// TIA Portal project "SCL" (V19)

(* hardware
DEVICE "S7-1500/ET200MP station_1"  S7-1500 station
   slot 0: "Rail_0"  Rack  6ES7 590-1***0-0AA0
   slot 1: "PLC_1"  CPU 1513-1 PN  6ES7 513-1AL02-0AB0  V2.9
      slot 3: "CPU display_1"  6ES7591-1AA00-0AA0
      slot 32768: "PROFINET interface_1"  X1
         slot 32769: "Port_1"  X1 P1
         slot 32770: "Port_2"  X1 P2
      slot 34817: "Virtual CP interface port_1"  Virtual CP interface port  Virtual CP interface port
   slot 2: "DI 16x24VDC BA_1"  DI 16x24VDC BA  6ES7 521-1BH10-0AA0  V1.1
   slot 3: "DQ 16x24VDC/0.5A BA_1"  DQ 16x24VDC/0.5A BA  6ES7 522-1BH10-0AA0  V1.1
*)

// ===== PLC "PLC_1"  CPU 1513-1 PN =====

VAR_GLOBAL   // PLC tag table "Default tag table"
   "At Entry" AT %I0.0 : Bool;
   "At Load" AT %I0.1 : Bool;
   "At left" AT %I0.2 : Bool;
   "At Middle" AT %I0.3 : Bool;
   "At Right" AT %I0.4 : Bool;
   "At Unload" AT %I0.5 : Bool;
   "At Exit" AT %I0.6 : Bool;
   "Moving X" AT %I0.7 : Bool;
   "Moving Z" AT %I1.0 : Bool;
   "Start" AT %I1.1 : Bool;
   "Reset" AT %I1.2 : Bool;
   "Stop" AT %I1.3 : Bool;
   "Emergency stop" AT %I1.4 : Bool;
   "Auto" AT %I1.5 : Bool;
   "FACTORY I/O (Runing)" AT %I1.6 : Bool;
   "Entry Conveyor" AT %Q0.0 : Bool;
   "Load Conveyor" AT %Q0.1 : Bool;
   "Forks Left" AT %Q0.2 : Bool;
   "Forks Right" AT %Q0.3 : Bool;
   "Lift" AT %Q0.4 : Bool;
   "Unload Conveyor" AT %Q0.5 : Bool;
   "Exit Conveyor" AT %Q0.6 : Bool;
   "Start light" AT %Q0.7 : Bool;
   "Reset light" AT %Q1.0 : Bool;
   "Stop light" AT %Q1.1 : Bool;
   "Target position" AT %QW30 : Int;
   "State0" AT %M0.0 : Bool;
   "State1" AT %M0.1 : Bool;
   "State2" AT %M0.2 : Bool;
   "State3" AT %M0.3 : Bool;
   "State4" AT %M0.4 : Bool;
   "State5" AT %M0.5 : Bool;
   "State6" AT %M0.6 : Bool;
   "State7" AT %M0.7 : Bool;
   "State8" AT %M1.0 : Bool;
   "State9" AT %M1.1 : Bool;
   "Tag_1" AT %M1.3 : Bool;
   "Tag_2" AT %M1.4 : Bool;
   "Tag_3" AT %M1.5 : Bool;
   "Tag_4" AT %M1.6 : Bool;
   "Tag_5" AT %M1.2 : Bool;
   "t" AT %MW30 : Int;
   "Tag_6" AT %M1.7 : Bool;
   "case" AT %MW2 : Int;
END_VAR

FUNCTION "Block_1" : Void   // FC1, SCL
{ S7_Optimized_Access := 'TRUE' }
VERSION : 0.1
BEGIN
   IF "Start light" THEN

       // Statement section IF
       CASE "case" OF
           0:  // Statement section case 1
               "Entry Conveyor" := FALSE;
               "Load Conveyor" := FALSE;
               "Forks Left" := FALSE;
               "Forks Right" := FALSE;
               "Lift" := FALSE;
               "Unload Conveyor" := FALSE;
               "Exit Conveyor" := FALSE;
               "case" := 1;

           1:  // Statement section case 2 to 4
               "Entry Conveyor" := TRUE;
               "Load Conveyor" := TRUE;
               IF NOT "At Load" THEN
                   // Statement section IF
                   "case" := 2;
               END_IF;
           2:
               "Forks Left" := 1;
               "Entry Conveyor" := 0;
               "Load Conveyor" := 0;
               IF "At left" THEN
                   // Statement section IF
                   "case" := 3;
               END_IF;
           3:
               "Lift" := 1;
               "R_TRIG_DB"(CLK:="Moving Z",
                           Q=>"Tag_1");

               IF "Tag_1" THEN
                   // Statement section IF
                   "case" := 4;
               END_IF;

           4:
               "Forks Left" := 0;
               IF "At Middle" THEN
                   // Statement section IF
                   "case" := 5;
               END_IF;
               "Tag_5" := 1;
           5:


               //"R_TRIG_DB_1"(CLK:="Tag_5",
                             //Q=>"Tag_6");
               //IF "Tag_5" THEN
                   // Statement section IF
                  // "Tag_5" := FALSE;
                  // "Target position" := "t";
                  // "t" := "t" + 1;


              // END_IF;
               WHILE "Tag_5" DO
                   // Statement section WHILE
                   "Tag_5" := FALSE;
                   "Target position" := "t";
                   "t" := "t" + 1;;
               END_WHILE;



               "F_TRIG_DB"(CLK:="Moving Z",
                           Q=>"Tag_2");

               "F_TRIG_DB_1"(CLK:="Moving X",
                             Q=>"Tag_3");

               IF ("Tag_2" AND NOT "Moving X") OR ("Tag_3" AND NOT "Moving Z") THEN
                   // Statement section IF

                   "case":=6;
               END_IF;

           6:

               "Forks Right" := 1;
               IF "At Right" THEN
                   // Statement section IF
                   "case" := 7;
               END_IF;
           7:
               "Lift" := 0
               ;
               "F_TRIG_DB_2"(CLK:="Moving Z",
                             Q=>"Tag_4");
               IF "Tag_4" THEN
                   // Statement section IF
                   "case" := 8;
               END_IF;
           8:
               "Forks Right" := 0;
               IF "At Middle" THEN
                   // Statement section IF
                   "case":=9;
               END_IF;
           9:
               "Target position" := 55;
               "case" := 0;


       END_CASE;

       ;
   END_IF;
END_FUNCTION

FUNCTION "Block_2" : Void   // FC2, LAD
{ S7_Optimized_Access := 'TRUE' }
VERSION : 0.1
BEGIN

REGION Network 1
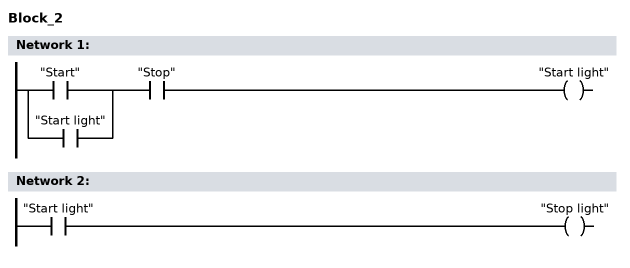
   RUNG wire#powerrail
      Contact( "Start" )
      wire#w1
      Contact( "Stop" )
      Coil( "Start light" )
   END_RUNG
   RUNG wire#powerrail
      Contact( "Start light" )
   END_RUNG wire#w1
   // the same network as SCL:
   "Start light" := ("Start" OR "Start light") AND "Stop";
END_REGION

REGION Network 2
   RUNG wire#powerrail
      Contact( "Start light" )
      Coil( "Stop light" )
   END_RUNG
   // the same network as SCL:
   "Stop light" := "Start light";
END_REGION
END_FUNCTION

ORGANIZATION_BLOCK "Main"   // OB1, LAD, ProgramCycle
TITLE = "Main Program Sweep (Cycle)"
{ S7_Optimized_Access := 'TRUE' }
VERSION : 0.1
   VAR_INPUT
      Initial_Call : Bool;   // Initial call of this OB
      Remanence : Bool;   // =True, if remanent data are available
   END_VAR
BEGIN

REGION Network 1
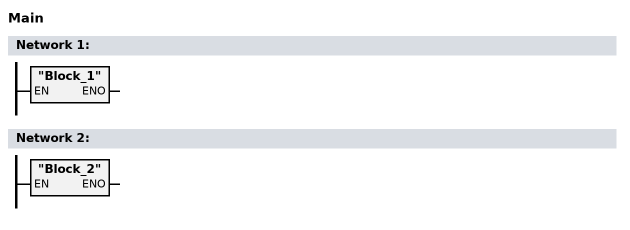
   RUNG wire#powerrail
      "Block_1"()
   END_RUNG
   // the same network as SCL:
   "Block_1"();
END_REGION

REGION Network 2
   RUNG wire#powerrail
      "Block_2"()
   END_RUNG
   // the same network as SCL:
   "Block_2"();
END_REGION
END_ORGANIZATION_BLOCK

ORGANIZATION_BLOCK "Startup"   // OB100, LAD, Startup
TITLE = "Complete Restart"
{ S7_Optimized_Access := 'TRUE' }
VERSION : 0.1
   VAR_INPUT
      LostRetentive : Bool;   // True if retentive data are lost
      LostRTC : Bool;   // True if date and time are lost
   END_VAR
BEGIN

REGION Network 1
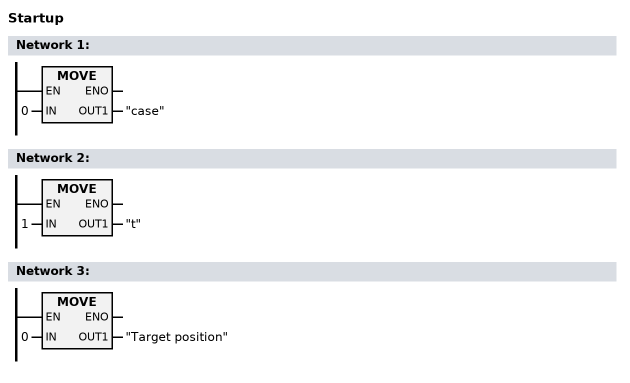
   RUNG wire#powerrail
      Move(in := 0, out1 => "case")
   END_RUNG
   // the same network as SCL:
   "case" := 0;
END_REGION

REGION Network 2
   RUNG wire#powerrail
      Move(in := 1, out1 => "t")
   END_RUNG
   // the same network as SCL:
   "t" := 1;
END_REGION

REGION Network 3
   RUNG wire#powerrail
      Move(in := 0, out1 => "Target position")
   END_RUNG
   // the same network as SCL:
   "Target position" := 0;
END_REGION
END_ORGANIZATION_BLOCK